// TIA Portal V20 export
DATA_BLOCK "CallEquipment_DB"   // DB169
{ DB_Accessible_From_OPC_UA := 'FALSE' }
// stored: AssignedProDiagFB Unit1.Em4.ProDiag, DBAccessibleFromOPCUA false, DBAccessibleFromWebserver false, InstanceOfName Unit1.Em4.CallEquipment, InstanceOfType FB, Namespace Unit1.Em4
"Unit1.Em4.CallEquipment"
   // VAR_INPUT
   //    ZoneOperationEnable { ExternalWritable := 'False'} : "LWONIK_typeSafetyZoneManualOperation";
   // END_VAR
   // VAR_IN_OUT
   //    unitStatus : "LAF_typeUnitStatus";
   //    emFeedback : "LUC_typeEmFeedback";
   //    unitAlarmDB : "LAF_typeAlarms";
   // END_VAR
   // VAR
   //    InstSequenceSideTapeLoading { ExternalWritable := 'False'} : "Unit1.Em4.Sequence_1_SideTapeLoading";
   //    InstSequenceSideTapeAttachment { ExternalWritable := 'False'} : "Unit1.Em4.Sequence_2_SideTapeAttachment";
   //    InstSequenceSideTapeFixStage { ExternalWritable := 'False'} : "Unit1.Em4.Sequence_3_SideTapeFixStage";
   //    instSideTapeLoadingHomeJob1 { ExternalWritable := 'False'} : "LAF_SelectJob";
   //    instSideTapeLoadingChargeJob2 { ExternalWritable := 'False'} : "LAF_SelectJob";
   //    instSideTapeAttachHomeJob1 { ExternalWritable := 'False'} : "LAF_SelectJob";
   //    instSideTapeAttachRightTapeGetJob2 { ExternalWritable := 'False'} : "LAF_SelectJob";
   //    instSideTapeAttachLeftTapeGetJob3 { ExternalWritable := 'False'} : "LAF_SelectJob";
   //    instSideTapeAttachTape1PutJob4 { ExternalWritable := 'False'} : "LAF_SelectJob";
   //    instSideTapeAttachTape2PutJob5 { ExternalWritable := 'False'} : "LAF_SelectJob";
   //    instSideTapeAttachTape3PutJob6 { ExternalWritable := 'False'} : "LAF_SelectJob";
   //    instSideTapeAttachTape4PutJob7 { ExternalWritable := 'False'} : "LAF_SelectJob";
   //    instSideTapeAttachTapeIdleJob8 { S7_SetPoint := 'True'} : "LAF_SelectJob";
   //    instSideTapeFixStageHomeJob1 { ExternalWritable := 'False'} : "LAF_SelectJob";
   //    instSideTapeFixStageLoadJob2 { ExternalWritable := 'False'} : "LAF_SelectJob";
   //    instSideTapeFixStageTaping1Job3 { ExternalWritable := 'False'} : "LAF_SelectJob";
   //    instSideTapeFixStageTaping2Job4 { ExternalWritable := 'False'} : "LAF_SelectJob";
   //    instSideTapeFixStageTaping3Job5 { ExternalWritable := 'False'} : "LAF_SelectJob";
   //    instSideTapeFixStageTaping4Job6 { ExternalWritable := 'False'} : "LAF_SelectJob";
   //    instSideTapeFixStageUnloadJob7 { ExternalWritable := 'False'} : "LAF_SelectJob";
   //    instCmSideTapeSafetyPin { ExternalWritable := 'False'} : "LBC_DigitalSignalCn";
   //    instCmSideTapeJRDetect { ExternalWritable := 'False'} : "LBC_DigitalSignalCn";
   //    instCmSideTapeDiameter { ExternalWritable := 'False'} : "LBC_DigitalSignalCn";
   //    instCmSideTapeFixStageAxisX { ExternalWritable := 'False'} : "LBC_Axis64Pos_TecPlcCn";
   //    instCmSideTapeFixStageAxisC { ExternalWritable := 'False'} : "LBC_Axis64Pos_TecPlcCn";
   //    instCmSideTapeAttachmentAxisX { ExternalWritable := 'False'} : "LBC_Axis64Pos_TecPlcCn";
   //    instCmSideTapeAttachmentAxisY { ExternalWritable := 'False'} : "LBC_Axis64Pos_TecPlcCn";
   //    instCmSideTapeLoadingBwdFwd { ExternalWritable := 'False'} : "LBC_TwoWayActuatorCn";
   //    instCmSideTapeLoadingClampOpenClose { ExternalWritable := 'False'} : "LBC_TwoWayActuatorCn";
   //    instCmSideTapeCutterBwdFwd { ExternalWritable := 'False'} : "LBC_TwoWayActuatorCn";
   //    instCmSideTapeCutterClampBwdFwd { ExternalWritable := 'False'} : "LBC_TwoWayActuatorCn";
   //    instCmSideTapeTensionBwdFwd { ExternalWritable := 'False'} : "LBC_TwoWayActuatorCn";
   //    instCmSideTapeAttachmentLeftBwdFwd { ExternalWritable := 'False'} : "LBC_TwoWayActuatorCn";
   //    instCmSideTapeAttachmentRightBwdFwd { ExternalWritable := 'False'} : "LBC_TwoWayActuatorCn";
   //    instCmSideTapeAttachmentBtmBwdFwd { ExternalWritable := 'False'} : "LBC_TwoWayActuatorCn";
   //    instCmSideTapeFixStageClampOpenClose { ExternalWritable := 'False'} : "LBC_TwoWayActuatorCn";
   //    instCmSideTapeAttachment1TopVaccumOffOn { ExternalWritable := 'False'} : "LBC_TwoWayActuatorCn";
   //    instCmSideTapeAttachment1BtmVaccumOffOn { ExternalWritable := 'False'} : "LBC_TwoWayActuatorCn";
   //    instCmSideTapeAttachment2TopVaccumOffOn { ExternalWritable := 'False'} : "LBC_TwoWayActuatorCn";
   //    instCmSideTapeAttachment2BtmVaccumOffOn { ExternalWritable := 'False'} : "LBC_TwoWayActuatorCn";
   //    instQrHandyReader { ExternalWritable := 'False'} : "LER_QRread_DM8700";
   //    instInterlockSideTapeFixStageAxisX { ExternalWritable := 'False'} : "LER_Axis64Pos_InterlockSummary";
   //    instInterlockSideTapeFixStageAxisC { ExternalWritable := 'False'} : "LER_Axis64Pos_InterlockSummary";
   //    instInterlockSideTapeAttachmentAxisX { ExternalWritable := 'False'} : "LER_Axis64Pos_InterlockSummary";
   //    instInterlockSideTapeAttachmentAxisY { ExternalWritable := 'False'} : "LER_Axis64Pos_InterlockSummary";
   //    instEventsPFE { ExternalWritable := 'False'} : "Unit1.Em4.EventsPFE";
   //    instManageAlarms { ExternalWritable := 'False'} : "LAF_ManageAlarms";
   //    statUnitStatus { ExternalWritable := 'False'} : "LAF_typeUnitStatus";
   //    statSlmStatus { ExternalWritable := 'False'} : Struct
   //       running : Bool;
   //       powerOff : Bool;
   //    END_STRUCT;
   //    statTonTime { ExternalWritable := 'False'} : Array[0..999] of TON_TIME;
   //    statTofTime { ExternalWritable := 'False'} : Array[0..9] of TOF_TIME;
   //    statPulse { ExternalWritable := 'False'} : Array[0..999] of Bool;
   //    statPartData { ExternalWritable := 'False'} : "LER_typePartData";
   //    statEnableManualCmds { ExternalWritable := 'False'} : Bool;
   //    SideTapeIdleCondition : Bool;
   //    "*** Interlock Axis ***" : Bool;
   //    sideTapeFixStageAxisX_JogCW { S7_SetPoint := 'True'} : "LER_Axis_Jog";
   //    sideTapeFixStageAxisX_JogCCW { S7_SetPoint := 'True'} : "LER_Axis_Jog";
   //    sideTapeFixStageAxisC_JogCW { S7_SetPoint := 'True'} : "LER_Axis_Jog";
   //    sideTapeFixStageAxisC_JogCCW { S7_SetPoint := 'True'} : "LER_Axis_Jog";
   //    sideTapeAttachmentAxisX_JogCW { S7_SetPoint := 'True'} : "LER_Axis_Jog";
   //    sideTapeAttachmentAxisX_JogCCW { S7_SetPoint := 'True'} : "LER_Axis_Jog";
   //    sideTapeAttachmentAxisY_JogCW { S7_SetPoint := 'True'} : "LER_Axis_Jog";
   //    sideTapeAttachmentAxisY_JogCCW { S7_SetPoint := 'True'} : "LER_Axis_Jog";
   //    sideTapeFixStageAxisX_interlock { S7_SetPoint := 'True'} : Array[0..10] of "LER_Axis_Absolute";
   //    sideTapeFixStageAxisC_interlock { S7_SetPoint := 'True'} : Array[0..10] of "LER_Axis_Absolute";
   //    sideTapeAttachmentAxisX_interlock { S7_SetPoint := 'True'} : Array[0..15] of "LER_Axis_Absolute";
   //    sideTapeAttachmentAxisY_interlock { S7_SetPoint := 'True'} : Array[0..15] of "LER_Axis_Absolute";
   //    sideTapeFixStageAxisX_IntPos : Array[0..9] of Struct
   //       "Int" : Array[1..10] of Bool;
   //    END_STRUCT;
   //    sideTapeFixStageAxisC_IntPos : Array[0..9] of Struct
   //       "Int" : Array[1..10] of Bool;
   //    END_STRUCT;
   //    sideTapeAttachmentAxisX_IntPos : Array[0..15] of Struct
   //       "Int" : Array[1..10] of Bool;
   //    END_STRUCT;
   //    sideTapeAttachmentAxisY_IntPos : Array[0..15] of Struct
   //       "Int" : Array[1..10] of Bool;
   //    END_STRUCT;
   //    sideTapeFixStageAxisX_IntHome : Array[0..9] of Bool;
   //    sideTapeFixStageAxisC_IntHome : Array[0..9] of Bool;
   //    sideTapeAttachmentAxisX_IntHome : Array[0..15] of Bool;
   //    sideTapeAttachmentAxisY_IntHome : Array[0..15] of Bool;
   //    "sideTapeFixStageAxisX PosAbsolute" : Array[0..10] of Bool;
   //    SideTapeFixStageAxisC_PosAbsolute : Array[0..10] of Bool;
   //    sideTapeAttachmentAxisX_PosAbsolute : Array[0..15] of Bool;
   //    sideTapeAttachmentAxisY_PosAbsolute : Array[0..15] of Bool;
   //    sideTapeFixStageAxisX_Home { S7_SetPoint := 'True'} : "LER_Axis_Homing";
   //    SideTapeFixStageAxisC_Home { S7_SetPoint := 'True'} : "LER_Axis_Homing";
   //    sideTapeAttachmentAxisX_Home { S7_SetPoint := 'True'} : "LER_Axis_Homing";
   //    sideTapeAttachmentAxisY_Home { S7_SetPoint := 'True'} : "LER_Axis_Homing";
   //    "*** Interlock TwoWay ***" { S7_SetPoint := 'True'} : "LER_Axis_Homing";
   //    instCmSideTapeLoadingDownUpInterlock { S7_SetPoint := 'True'} : Array[0..2] of "LER_Actuator";
   //    instCmSideTapeLoadingClampOpenCloseInterlock { S7_SetPoint := 'True'} : Array[0..2] of "LER_Actuator";
   //    instCmSideTapeCutterBwdFwdInterlock { S7_SetPoint := 'True'} : Array[0..2] of "LER_Actuator";
   //    instCmSideTapeCutterClampBwdFwdInterlock { S7_SetPoint := 'True'} : Array[0..2] of "LER_Actuator";
   //    instCmSideTapeTensionBwdFwdInterlock { S7_SetPoint := 'True'} : Array[0..2] of "LER_Actuator";
   //    instCmSideTapeAttachmentLeftBwdFwdInterlock { S7_SetPoint := 'True'} : Array[0..2] of "LER_Actuator";
   //    instCmSideTapeAttachmentRightBwdFwdInterlock { S7_SetPoint := 'True'} : Array[0..2] of "LER_Actuator";
   //    instCmSideTapeAttachmentBtmBwdFwdInterlock { S7_SetPoint := 'True'} : Array[0..2] of "LER_Actuator";
   //    instCmSideTapeFixStageClampOpenCloseInterlock { S7_SetPoint := 'True'} : Array[0..2] of "LER_Actuator";
   //    instCmSideTapeAttachment1TopVaccumOffOnInterlock { S7_SetPoint := 'True'} : Array[0..2] of "LER_Actuator";
   //    instCmSideTapeAttachment1BtmVaccumOffOnInterlock { S7_SetPoint := 'True'} : Array[0..2] of "LER_Actuator";
   //    instCmSideTapeAttachment2TopVaccumOffOnInterlock { S7_SetPoint := 'True'} : Array[0..2] of "LER_Actuator";
   //    instCmSideTapeAttachment2BtmVaccumOffOnInterlock { S7_SetPoint := 'True'} : Array[0..2] of "LER_Actuator";
   //    sideTapeLoadingDownUp_Inpos : Array[0..2] of Struct
   //       "Int" : Array[1..10] of Bool;
   //    END_STRUCT;
   //    sideTapeLoadingClampOpenClose_Inpos : Array[0..2] of Struct
   //       "Int" : Array[1..10] of Bool;
   //    END_STRUCT;
   //    sideTapeCutterBwdFwd_Inpos : Array[0..2] of Struct
   //       "Int" : Array[1..10] of Bool;
   //    END_STRUCT;
   //    sideTapeCutterClampBwdFwd_Inpos : Array[0..2] of Struct
   //       "Int" : Array[1..10] of Bool;
   //    END_STRUCT;
   //    sideTapeTensionBwdFwd_Inpos : Array[0..2] of Struct
   //       "Int" : Array[1..10] of Bool;
   //    END_STRUCT;
   //    sideTapeAttachmentLeftBwdFwd_Inpos : Array[0..2] of Struct
   //       "Int" : Array[1..10] of Bool;
   //    END_STRUCT;
   //    sideTapeAttachmentRightBwdFwd_Inpos : Array[0..2] of Struct
   //       "Int" : Array[1..10] of Bool;
   //    END_STRUCT;
   //    sideTapeAttachmentBtmBwdFwd_Inpos : Array[0..2] of Struct
   //       "Int" : Array[1..10] of Bool;
   //    END_STRUCT;
   //    sideTapeFixStageClampOpenClose_Inpos : Array[0..2] of Struct
   //       "Int" : Array[1..10] of Bool;
   //    END_STRUCT;
   //    sideTapeAttachment1TopVaccumOffOn_Inpos : Array[0..2] of Struct
   //       "Int" : Array[1..10] of Bool;
   //    END_STRUCT;
   //    sideTapeAttachment1BtmVaccumOffOn_Inpos : Array[0..2] of Struct
   //       "Int" : Array[1..10] of Bool;
   //    END_STRUCT;
   //    sideTapeAttachment2TopVaccumOffOn_Inpos : Array[0..2] of Struct
   //       "Int" : Array[1..10] of Bool;
   //    END_STRUCT;
   //    sideTapeAttachment2BtmVaccumOffOn_Inpos : Array[0..2] of Struct
   //       "Int" : Array[1..10] of Bool;
   //    END_STRUCT;
   //    citi_Ptrig : Array[0..20] of Bool;
   //    citiTon : Array[0..20] of TON_TIME;
   //    citi : Time;
   //    citiTest : Array[0..20] of Bool;
   // END_VAR
BEGIN
END_DATA_BLOCK
